Staubli VAL3: TeachSimu.pgx

public program TeachSimu(num x_nStart, num x_nEnd)
begin
  //示教或者调图时模拟
  //不需要进行读取文件




  call KillTask()
  setMoveId(0)
  nStartTraj=nEndTraj
  //DataBase:bSimuIO=false

  if TxtFile:bWeldEnable
    taskCreateSync "Preset",0.008,bSync,Preset()
    // taskCreateSync "WeldEnd",0.008,bSync,WeldEnd()

  else
    taskCreate "Preset",100,Preset()
  endIf

  if x_nEnd<=0 or x_nStart<=0
    taskCreate "Move",100,Move()
  else
     taskCreate "Move",100,PartMove(x_nStart,x_nEnd)
  endIf
  wait(DataBase:bMoveTask==false)
  //焊接的回退
  if (DataBase:nInterfaceType==13 or DataBase:nInterfaceType==6) and TxtFile:bWeldEnable
    DataBase:nInterfaceType=9
  endIf

end
